// Mitsubishi GX Works2 project: PLC_group7   PLC: FX3G

// global labels: Global1
VAR_GLOBAL
  Lamp10 AT Y010 : BOOL;
  Switch7 AT X007 : BOOL;
  D_OrangeInventory AT D1100 : REAL;
  D_ClemInventory AT D1102 : REAL;
  D_PomInventory AT D1104 : REAL;
END_VAR
VAR_GLOBAL CONSTANT
  K_Value2 : REAL := 2.0;
END_VAR
VAR_GLOBAL
  D_halfOrange_Start AT D1106 : REAL;
END_VAR
VAR_GLOBAL CONSTANT
  K_Value50 : REAL := 50.0;
END_VAR
VAR_GLOBAL
  D_Amount_CleOrPom_ToWash AT D1112 : REAL;
END_VAR
VAR_GLOBAL CONSTANT
  K_Value0 : REAL;
END_VAR
VAR_GLOBAL
  M_emptyInventory AT M0 : BOOL;
END_VAR
VAR_GLOBAL CONSTANT
  K_Value30int : INT := 30;
END_VAR
VAR_GLOBAL
  M_emergencySwitch AT M2 : BOOL;
  Switch10 AT X010 : BOOL;
  Switch2 AT X002 : BOOL;
  Lamp5 AT Y005 : BOOL;
  Timer_Wash AT TC2 : BOOL;
  Timer_Wash_Status AT TS2 : BOOL;
  D_Orange_WashVessel AT D1120 : REAL;
  D_Clem_WashVessel AT D1116 : REAL;
  D_Pom_WashVessel AT D1118 : REAL;
  D_Amount_Orange_ToWash AT D1114 : REAL;
  Lamp3 AT Y003 : BOOL;
  M_workDay AT M1 : BOOL;
  M_blinking AT M3 : BOOL;
  T_blink1 AT TC3 : BOOL;
  T_blink1_Status AT TS3 : BOOL;
  T_blink2 AT TC4 : BOOL;
  T_blink2_Status AT TS4 : BOOL;
  M_blinking_Light1 AT M10 : BOOL;
  M_blinking_Light2 AT M11 : BOOL;
  T_blinkingDuration AT TC5 : BOOL;
  T_blinkingDuration_Status AT TS5 : BOOL;
  D_SqueezeVessel AT D1122 : REAL;
  Lamp1 AT Y001 : BOOL;
  Switch1 AT X001 : BOOL;
  M_startSqueeze AT M12 : BOOL;
  Switch11 AT X011 : BOOL;
  Lamp2 AT Y002 : BOOL;
  C_squeeze AT CC0 : BOOL;
  C_squeeze_Status AT CS0 : BOOL;
END_VAR
VAR_GLOBAL CONSTANT
  K_Value2int : INT := 2;
END_VAR
VAR_GLOBAL
  T_squeeze AT TC6 : BOOL;
  T_squeeze_Status AT TS6 : BOOL;
  M_inputQuality AT M100 : BOOL;
  M_startBlink AT M5 : BOOL;
  M_startBlink_EndDay AT M6 : BOOL;
  M_startBlink_Squeeze AT M7 : BOOL;
  D_Juice AT D1124 : REAL;
  D_analogInput2 AT D8281 : INT;
  Switch3 AT X003 : BOOL;
END_VAR
VAR_GLOBAL CONSTANT
  K_Value405 : REAL := 405.5;
END_VAR
VAR_GLOBAL
  D_startOrange AT D1126 : REAL;
  D_startClem AT D1128 : REAL;
  D_startPom AT D1130 : REAL;
  D_qualityLevel AT D1224 : INT;
  D_qualityLevel2 AT D1226 : REAL;
END_VAR
VAR_GLOBAL CONSTANT
  K_Value2027 : REAL := 2027.5;
END_VAR
VAR_GLOBAL
  M_qualifiedJuice AT M13 : BOOL;
  T_qualityCheck AT TC7 : BOOL;
  T_qualityCheckStatus AT TS7 : BOOL;
  Lamp4 AT Y004 : BOOL;
  C_qualityCheck AT CC1 : BOOL;
  C_qualityCheck_Status AT CS1 : BOOL;
  M_squeezing AT M14 : BOOL;
  M_Check_mlay AT M200 : BOOL;
  D_start_min AT D1132 : REAL;
  D_output AT D8282 : INT;
END_VAR
VAR_GLOBAL CONSTANT
  K_Value15 : REAL := 15.0;
END_VAR
VAR_GLOBAL
  M_low_mlay AT M201 : BOOL;
  Lamp11 AT Y011 : BOOL;
  D_to_output AT D1134 : REAL;
  M_washed AT M300 : BOOL;
  M_collected AT M301 : BOOL;
  M_squeezed AT M302 : BOOL;
  M_checked AT M303 : BOOL;
  D_storage AT D1222 : REAL;
  M_updateStorage AT M15 : BOOL;
  D_amountToMake AT D1136 : REAL;
  D_halfOrange_Inventory AT D1138 : REAL;
  D_miniInventory AT D1136 : REAL;
END_VAR
VAR_GLOBAL CONSTANT
  K_Value0int : INT;
  K_Value5int : INT := 5;
  K_Value50int : INT := 50;
END_VAR
VAR_GLOBAL
  Switch0 AT X000 : BOOL;
END_VAR

// task Task_01 (event TRUE, interval 0, priority 31): POU_01

PROGRAM POU_01
(* structured ladder/FBD written out as ST: instructions are called as NAME(EN, inputs, outputs); _pN, _eN, _tN stand for wires *)
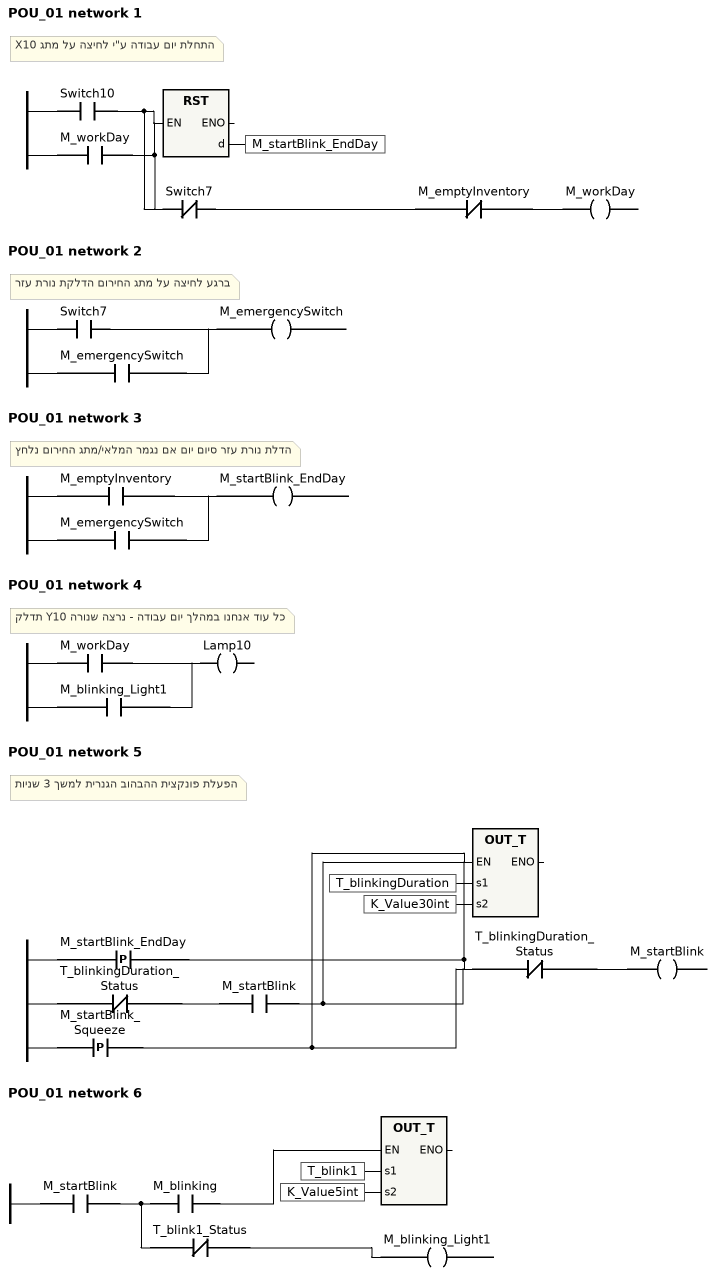
(* network 1 *)
(* התחלת יום עבודה ע"י לחיצה על מתג X10 *)
_p1 := Switch10 OR M_workDay;
M_workDay := _p1 AND NOT Switch7 AND NOT M_emptyInventory;
RST(_p1, M_startBlink_EndDay);
(* network 2 *)
(* ברגע לחיצה על מתג החירום הדלקת נורת עזר *)
M_emergencySwitch := Switch7 OR M_emergencySwitch;
(* network 3 *)
(* הדלת נורת עזר סיום יום אם נגמר המלאי/מתג החירום נלחץ *)
M_startBlink_EndDay := M_emptyInventory OR M_emergencySwitch;
(* network 4 *)
(* כל עוד אנחנו במהלך יום עבודה - נרצה שנורה Y10 תדלק *)
Lamp10 := M_workDay OR M_blinking_Light1;
(* network 5 *)
(* הפעלת פונקצית ההבהוב הגנרית למשך 3 שניות *)
_p1 := LDP(TRUE, M_startBlink_EndDay) OR (NOT T_blinkingDuration_Status AND M_startBlink) OR LDP(TRUE, M_startBlink_Squeeze);
OUT_T(_p1, T_blinkingDuration, K_Value30int);
M_startBlink := _p1 AND NOT T_blinkingDuration_Status;
(* network 6 *)
OUT_T(M_startBlink AND M_blinking, T_blink1, K_Value5int);
M_blinking_Light1 := M_startBlink AND NOT T_blink1_Status;
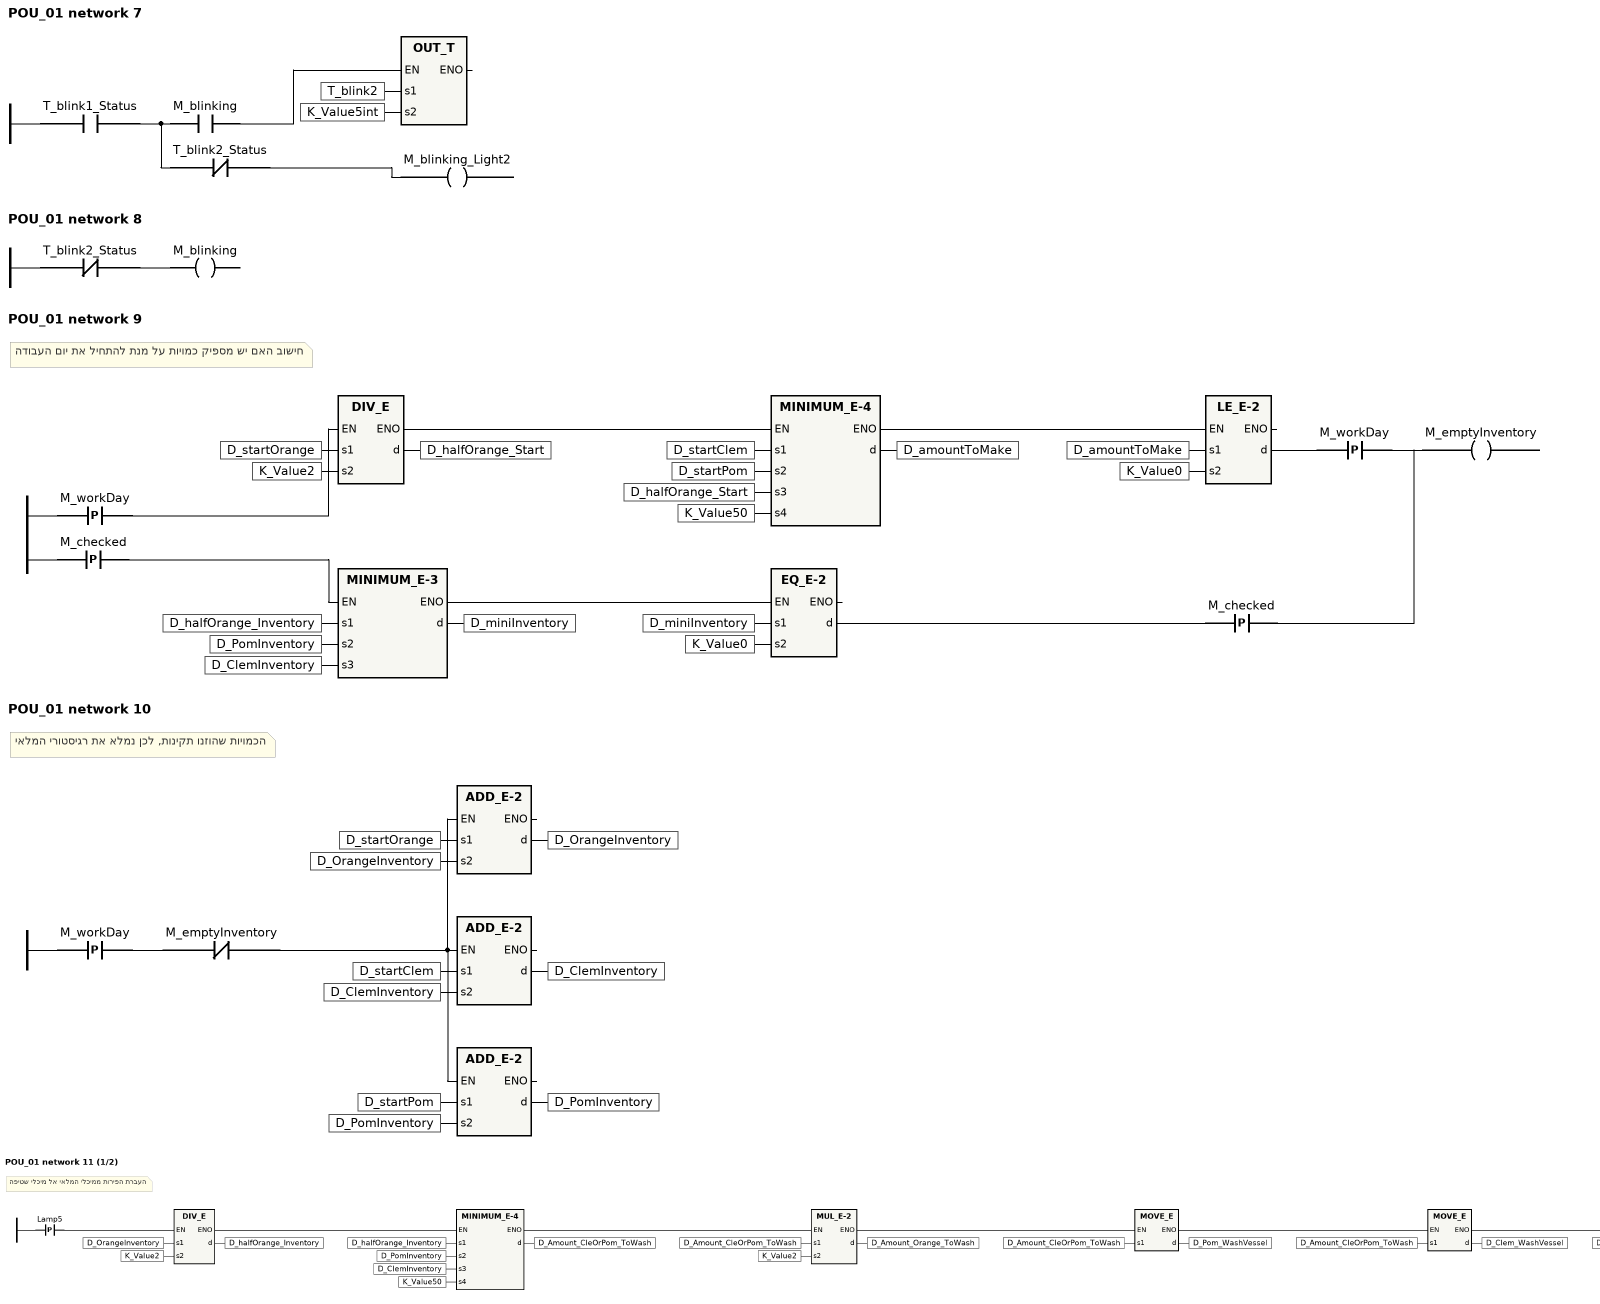
(* network 7 *)
OUT_T(T_blink1_Status AND M_blinking, T_blink2, K_Value5int);
M_blinking_Light2 := T_blink1_Status AND NOT T_blink2_Status;
(* network 8 *)
M_blinking := NOT T_blink2_Status;
(* network 9 *)
(* חישוב האם יש מספיק כמויות על מנת להתחיל את יום העבודה *)
_e1 := DIV_E(LDP(TRUE, M_workDay), D_startOrange, K_Value2, D_halfOrange_Start);
_e2 := MINIMUM_E(_e1, D_startClem, D_startPom, D_halfOrange_Start, K_Value50, D_amountToMake);
LE_E(_e2, D_amountToMake, K_Value0, _t3);
_e4 := MINIMUM_E(LDP(TRUE, M_checked), D_halfOrange_Inventory, D_PomInventory, D_ClemInventory, D_miniInventory);
EQ_E(_e4, D_miniInventory, K_Value0, _t5);
M_emptyInventory := (_t3 AND LDP(TRUE, M_workDay)) OR (_t5 AND LDP(TRUE, M_checked));
(* network 10 *)
(* הכמויות שהוזנו תקינות, לכן נמלא את רגיסטורי המלאי *)
_p1 := LDP(TRUE, M_workDay) AND NOT M_emptyInventory;
ADD_E(_p1, D_startOrange, D_OrangeInventory, D_OrangeInventory);
ADD_E(_p1, D_startClem, D_ClemInventory, D_ClemInventory);
ADD_E(_p1, D_startPom, D_PomInventory, D_PomInventory);
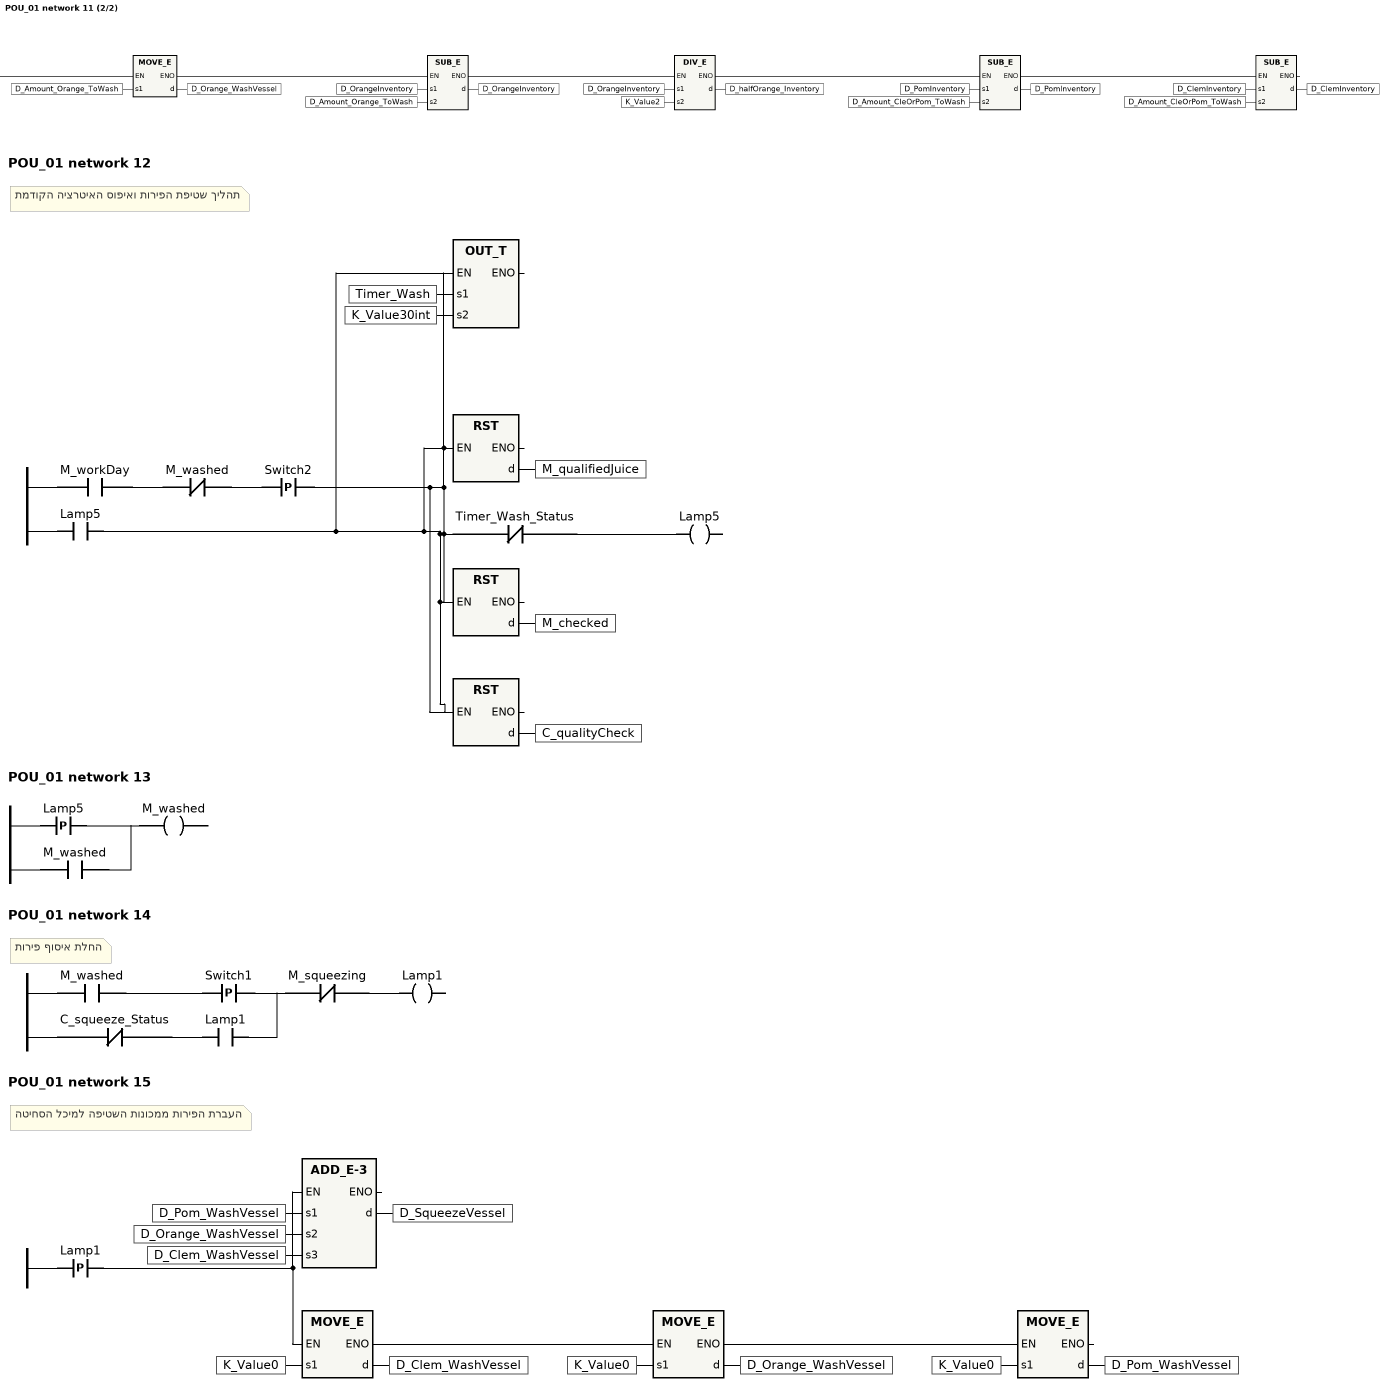
(* network 11 *)
(* העברת הפירות ממיכלי המלאי אל מיכלי שטיפה *)
_e1 := DIV_E(LDP(TRUE, Lamp5), D_OrangeInventory, K_Value2, D_halfOrange_Inventory);
_e2 := MINIMUM_E(_e1, D_halfOrange_Inventory, D_PomInventory, D_ClemInventory, K_Value50, D_Amount_CleOrPom_ToWash);
_e3 := MUL_E(_e2, D_Amount_CleOrPom_ToWash, K_Value2, D_Amount_Orange_ToWash);
_e4 := MOVE_E(_e3, D_Amount_CleOrPom_ToWash, D_Pom_WashVessel);
_e5 := MOVE_E(_e4, D_Amount_CleOrPom_ToWash, D_Clem_WashVessel);
_e6 := MOVE_E(_e5, D_Amount_Orange_ToWash, D_Orange_WashVessel);
_e7 := SUB_E(_e6, D_OrangeInventory, D_Amount_Orange_ToWash, D_OrangeInventory);
_e8 := DIV_E(_e7, D_OrangeInventory, K_Value2, D_halfOrange_Inventory);
_e9 := SUB_E(_e8, D_PomInventory, D_Amount_CleOrPom_ToWash, D_PomInventory);
SUB_E(_e9, D_ClemInventory, D_Amount_CleOrPom_ToWash, D_ClemInventory);
(* network 12 *)
(* תהליך שטיפת הפירות ואיפוס האיטרציה הקודמת *)
_p1 := (M_workDay AND NOT M_washed AND LDP(TRUE, Switch2)) OR Lamp5;
OUT_T(_p1, Timer_Wash, K_Value30int);
Lamp5 := _p1 AND NOT Timer_Wash_Status;
RST(_p1, M_qualifiedJuice);
RST(_p1, M_checked);
RST(_p1, C_qualityCheck);
(* network 13 *)
M_washed := LDP(TRUE, Lamp5) OR M_washed;
(* network 14 *)
(* החלת איסוף פירות *)
Lamp1 := ((M_washed AND LDP(TRUE, Switch1)) OR (NOT C_squeeze_Status AND Lamp1)) AND NOT M_squeezing;
(* network 15 *)
(* העברת הפירות ממכונות השטיפה למיכל הסחיטה *)
_p1 := LDP(TRUE, Lamp1);
ADD_E(_p1, D_Pom_WashVessel, D_Orange_WashVessel, D_Clem_WashVessel, D_SqueezeVessel);
_e2 := MOVE_E(_p1, K_Value0, D_Clem_WashVessel);
_e3 := MOVE_E(_e2, K_Value0, D_Orange_WashVessel);
MOVE_E(_e3, K_Value0, D_Pom_WashVessel);
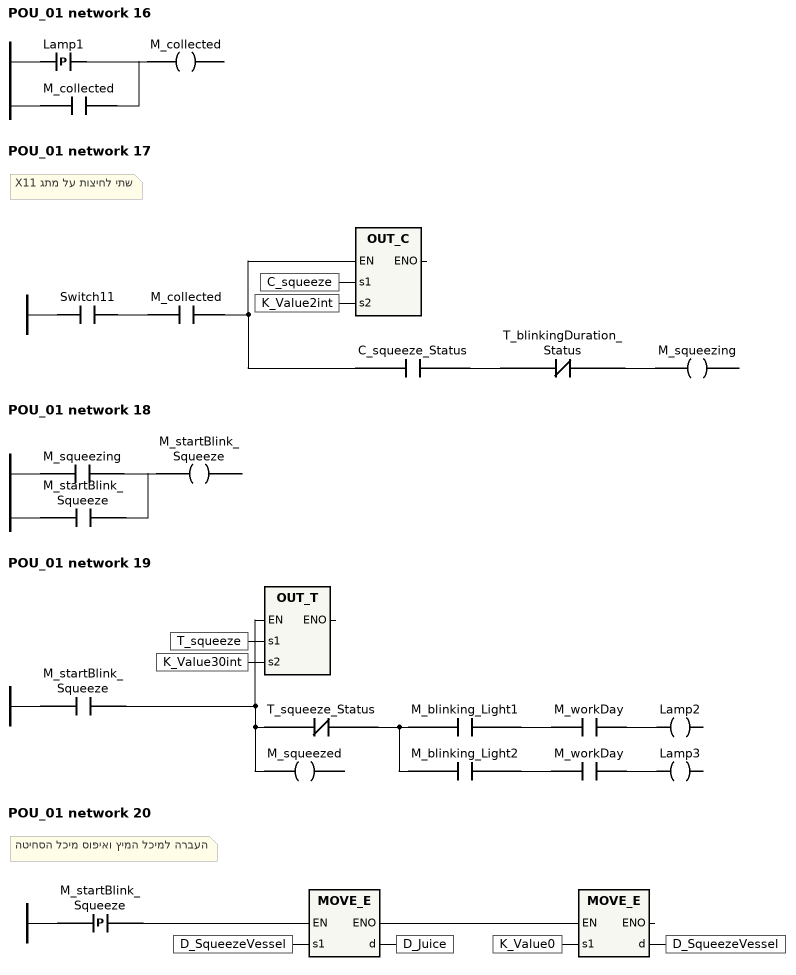
(* network 16 *)
M_collected := LDP(TRUE, Lamp1) OR M_collected;
(* network 17 *)
(* שתי לחיצות על מתג X11 *)
_p1 := Switch11 AND M_collected;
OUT_C(_p1, C_squeeze, K_Value2int);
M_squeezing := _p1 AND C_squeeze_Status AND NOT T_blinkingDuration_Status;
(* network 18 *)
M_startBlink_Squeeze := M_squeezing OR M_startBlink_Squeeze;
(* network 19 *)
OUT_T(M_startBlink_Squeeze, T_squeeze, K_Value30int);
_p1 := M_startBlink_Squeeze AND NOT T_squeeze_Status;
Lamp2 := _p1 AND M_blinking_Light1 AND M_workDay;
Lamp3 := _p1 AND M_blinking_Light2 AND M_workDay;
M_squeezed := M_startBlink_Squeeze;
(* network 20 *)
(* העברה למיכל המיץ ואיפוס מיכל הסחיטה *)
_e1 := MOVE_E(LDP(TRUE, M_startBlink_Squeeze), D_SqueezeVessel, D_Juice);
MOVE_E(_e1, K_Value0, D_SqueezeVessel);
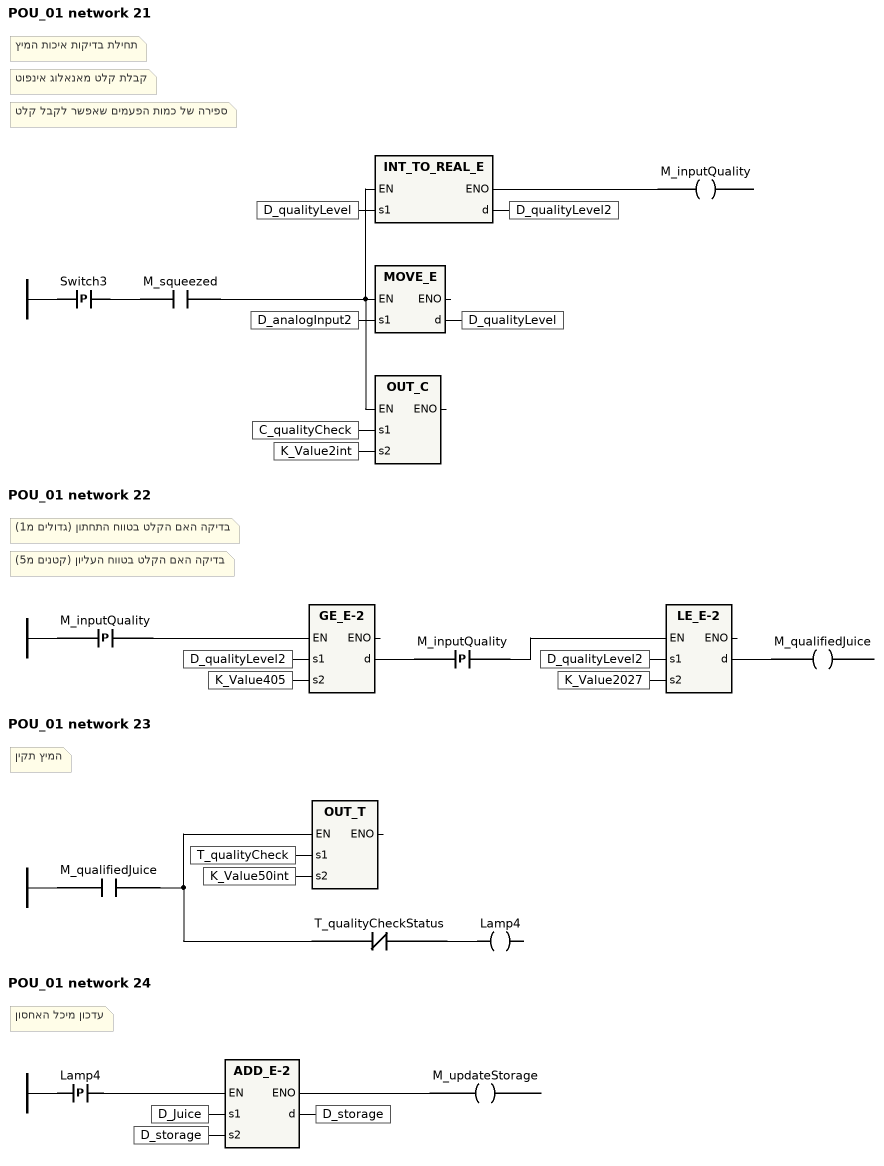
(* network 21 *)
(* תחילת בדיקות איכות המיץ *)
(* קבלת קלט מאנאלוג אינפוט *)
(* ספירה של כמות הפעמים שאפשר לקבל קלט *)
_p1 := LDP(TRUE, Switch3) AND M_squeezed;
MOVE_E(_p1, D_analogInput2, D_qualityLevel);
OUT_C(_p1, C_qualityCheck, K_Value2int);
_e2 := INT_TO_REAL_E(_p1, D_qualityLevel, D_qualityLevel2);
M_inputQuality := _e2;
(* network 22 *)
(* בדיקה האם הקלט בטווח התחתון (גדולים מ1) *)
(* בדיקה האם הקלט בטווח העליון (קטנים מ5) *)
GE_E(LDP(TRUE, M_inputQuality), D_qualityLevel2, K_Value405, _t1);
LE_E(_t1 AND LDP(TRUE, M_inputQuality), D_qualityLevel2, K_Value2027, _t2);
M_qualifiedJuice := _t2;
(* network 23 *)
(* המיץ תקין *)
OUT_T(M_qualifiedJuice, T_qualityCheck, K_Value50int);
Lamp4 := M_qualifiedJuice AND NOT T_qualityCheckStatus;
(* network 24 *)
(* עדכון מיכל האחסון *)
_e1 := ADD_E(LDP(TRUE, Lamp4), D_Juice, D_storage, D_storage);
M_updateStorage := _e1;
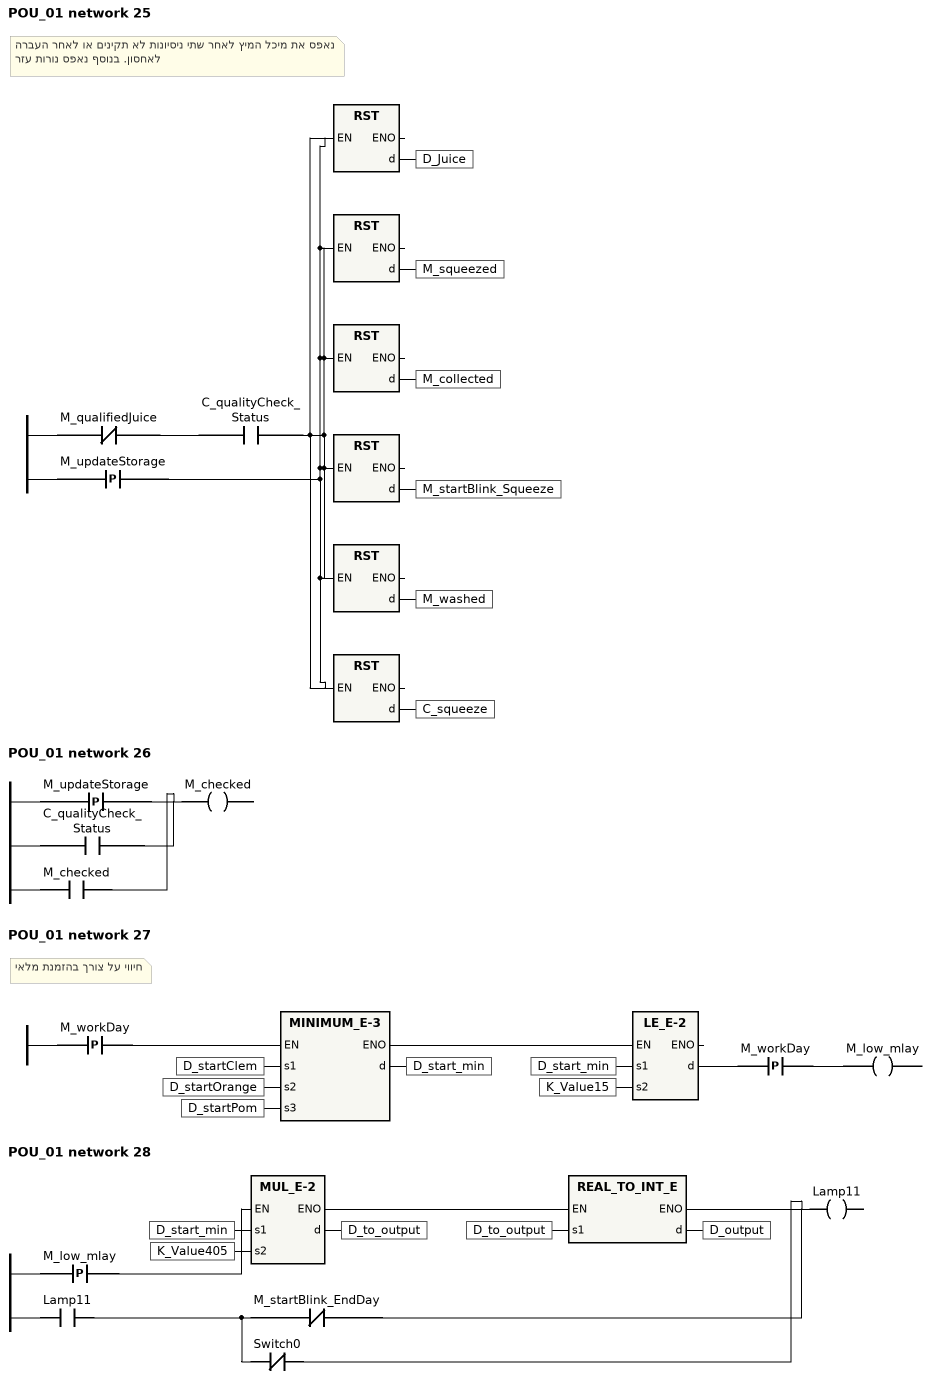
(* network 25 *)
(* נאפס את מיכל המיץ לאחר שתי ניסיונות לא תקינים או לאחר העברה לאחסון. בנוסף נאפס נורות עזר *)
_p1 := (NOT M_qualifiedJuice AND C_qualityCheck_Status) OR LDP(TRUE, M_updateStorage);
RST(_p1, D_Juice);
RST(_p1, M_squeezed);
RST(_p1, M_collected);
RST(_p1, M_startBlink_Squeeze);
RST(_p1, M_washed);
RST(_p1, C_squeeze);
(* network 26 *)
M_checked := LDP(TRUE, M_updateStorage) OR C_qualityCheck_Status OR M_checked;
(* network 27 *)
(* חיווי על צורך בהזמנת מלאי *)
_e1 := MINIMUM_E(LDP(TRUE, M_workDay), D_startClem, D_startOrange, D_startPom, D_start_min);
LE_E(_e1, D_start_min, K_Value15, _t2);
M_low_mlay := _t2 AND LDP(TRUE, M_workDay);
(* network 28 *)
_e1 := MUL_E(LDP(TRUE, M_low_mlay), D_start_min, K_Value405, D_to_output);
_e2 := REAL_TO_INT_E(_e1, D_to_output, D_output);
Lamp11 := _e2 OR (Lamp11 AND NOT M_startBlink_EndDay) OR (Lamp11 AND NOT Switch0);
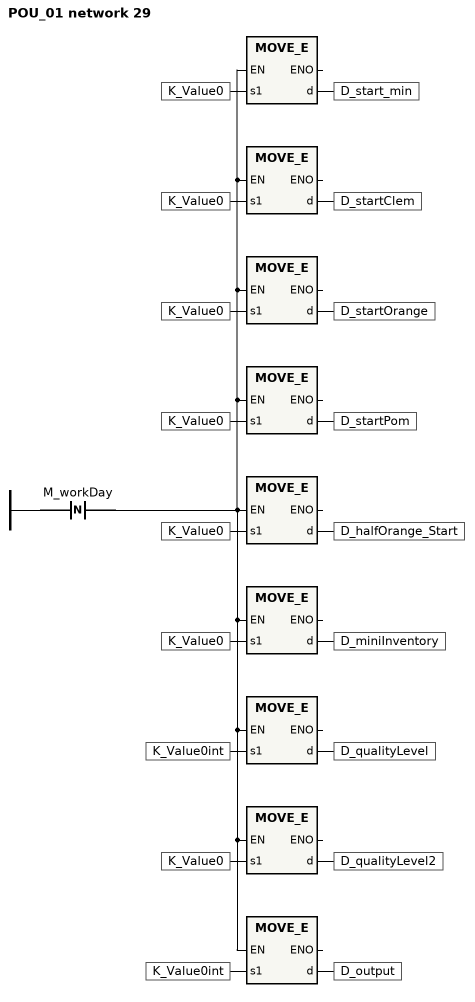
(* network 29 *)
_p1 := LDF(TRUE, M_workDay);
MOVE_E(_p1, K_Value0, D_start_min);
MOVE_E(_p1, K_Value0, D_startClem);
MOVE_E(_p1, K_Value0, D_startOrange);
MOVE_E(_p1, K_Value0, D_startPom);
MOVE_E(_p1, K_Value0, D_halfOrange_Start);
MOVE_E(_p1, K_Value0, D_miniInventory);
MOVE_E(_p1, K_Value0int, D_qualityLevel);
MOVE_E(_p1, K_Value0, D_qualityLevel2);
MOVE_E(_p1, K_Value0int, D_output);
END_PROGRAM
